{attribute addProperty BoxType "EL2595-0000-0019"}
{attribute addProperty Id "StatusAT %I*Status_214777E6162"}
{attribute addProperty CRC "2514413500"}
{attribute addProperty SizeInBites "16"}
{attribute addProperty SizeInBytes "2"}
TYPE DOX_Status_95DEE7BC :
STRUCT
	{attribute addProperty Name "Status"}
	Status AT %I* : Status_214777E6;
END_STRUCT
END_TYPE

(* stored: Version 1.2.0.0, ProductVersion 3.1.4024.9
   DUT DOX_Status_95DEE7BC: Id {a93782c3-1a84-45ce-84f7-c12a16e42028} *)
